// TIA Portal V20 export
FUNCTION_BLOCK "F-FB_Laser"   // FB140, F_LAD
{ S7_Optimized_Access := 'TRUE' }
// stored: AutoNumber false
   VAR
      FDBACK_LaserPowerSupply : FDBACK;
      FDBACK_Shutter : FDBACK;
      sFeedBackShutter : Bool;
      sAckFdbShutter : Bool;
      sLaserSupplyPower : Bool;
      sAckFdbPowLaser : Bool;
      sPositiveFrontButtonShutter : Bool;
      sNegativeFrontMaintenanceDoor : Bool;
      sNegativeFrontDoor : Bool;
      sNegativeRoofLeftDoor : Bool;
      sNegativeRoofRightDoor : Bool;
      sNegativeLaserExternDoor : Bool;
      sNegativeSasOneDoor : Bool;
   END_VAR
   VAR_TEMP   // added for the SCL form of the ladder/FBD networks
      _w1 : Bool;
      _w2 : Bool;
      _w3 : Bool;
      _w4 : Bool;
      _w5 : Bool;
      _w6 : Bool;
      _w7 : Bool;
   END_VAR
BEGIN

REGION Network 1: Laser shutter setting mode, allow opening shutter
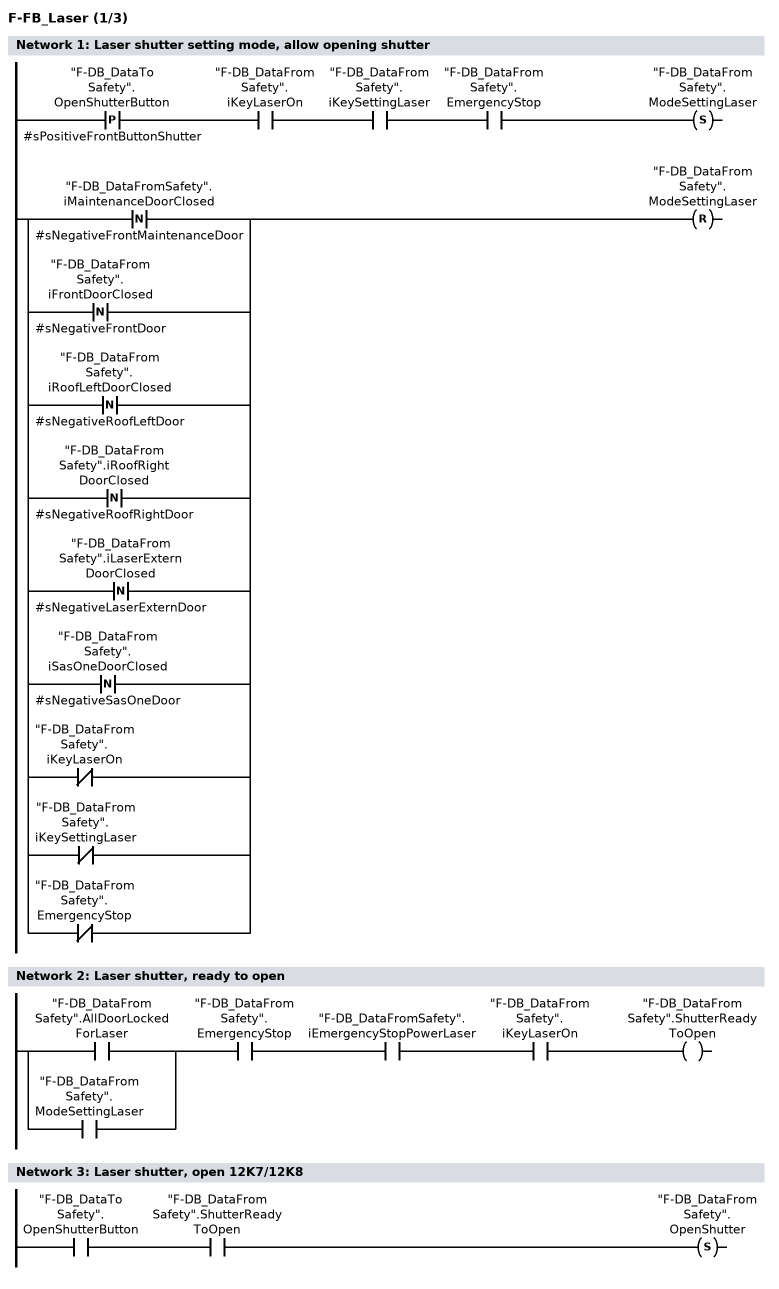
   RUNG wire#powerrail
      P_Contact(operand := "F-DB_DataToSafety".OpenShutterButton, bit := #sPositiveFrontButtonShutter)
      Contact( "F-DB_DataFromSafety".iKeyLaserOn )
      Contact( "F-DB_DataFromSafety".iKeySettingLaser )
      Contact( "F-DB_DataFromSafety".EmergencyStop )
      S_Coil( "F-DB_DataFromSafety".ModeSettingLaser )
   END_RUNG
   RUNG wire#powerrail
      N_Contact(operand := "F-DB_DataFromSafety".iMaintenanceDoorClosed, bit := #sNegativeFrontMaintenanceDoor)
      wire#w1
      R_Coil( "F-DB_DataFromSafety".ModeSettingLaser )
   END_RUNG
   RUNG wire#powerrail
      N_Contact(operand := "F-DB_DataFromSafety".iFrontDoorClosed, bit := #sNegativeFrontDoor)
   END_RUNG wire#w1
   RUNG wire#powerrail
      N_Contact(operand := "F-DB_DataFromSafety".iRoofLeftDoorClosed, bit := #sNegativeRoofLeftDoor)
   END_RUNG wire#w1
   RUNG wire#powerrail
      N_Contact(operand := "F-DB_DataFromSafety".iRoofRightDoorClosed, bit := #sNegativeRoofRightDoor)
   END_RUNG wire#w1
   RUNG wire#powerrail
      N_Contact(operand := "F-DB_DataFromSafety".iLaserExternDoorClosed, bit := #sNegativeLaserExternDoor)
   END_RUNG wire#w1
   RUNG wire#powerrail
      N_Contact(operand := "F-DB_DataFromSafety".iSasOneDoorClosed, bit := #sNegativeSasOneDoor)
   END_RUNG wire#w1
   RUNG wire#powerrail
      I_Contact( "F-DB_DataFromSafety".iKeyLaserOn )
   END_RUNG wire#w1
   RUNG wire#powerrail
      I_Contact( "F-DB_DataFromSafety".iKeySettingLaser )
   END_RUNG wire#w1
   RUNG wire#powerrail
      I_Contact( "F-DB_DataFromSafety".EmergencyStop )
   END_RUNG wire#w1
   // the same network as SCL:
   #_w1 := "F-DB_DataToSafety".OpenShutterButton AND NOT #sPositiveFrontButtonShutter;   // rising edge of "F-DB_DataToSafety".OpenShutterButton
   #sPositiveFrontButtonShutter := "F-DB_DataToSafety".OpenShutterButton;
   IF #_w1 AND "F-DB_DataFromSafety".iKeyLaserOn AND "F-DB_DataFromSafety".iKeySettingLaser AND "F-DB_DataFromSafety".EmergencyStop THEN
       "F-DB_DataFromSafety".ModeSettingLaser := TRUE;
   END_IF;
   #_w2 := NOT "F-DB_DataFromSafety".iMaintenanceDoorClosed AND #sNegativeFrontMaintenanceDoor;   // falling edge of "F-DB_DataFromSafety".iMaintenanceDoorClosed
   #sNegativeFrontMaintenanceDoor := "F-DB_DataFromSafety".iMaintenanceDoorClosed;
   #_w3 := NOT "F-DB_DataFromSafety".iFrontDoorClosed AND #sNegativeFrontDoor;   // falling edge of "F-DB_DataFromSafety".iFrontDoorClosed
   #sNegativeFrontDoor := "F-DB_DataFromSafety".iFrontDoorClosed;
   #_w4 := NOT "F-DB_DataFromSafety".iRoofLeftDoorClosed AND #sNegativeRoofLeftDoor;   // falling edge of "F-DB_DataFromSafety".iRoofLeftDoorClosed
   #sNegativeRoofLeftDoor := "F-DB_DataFromSafety".iRoofLeftDoorClosed;
   #_w5 := NOT "F-DB_DataFromSafety".iRoofRightDoorClosed AND #sNegativeRoofRightDoor;   // falling edge of "F-DB_DataFromSafety".iRoofRightDoorClosed
   #sNegativeRoofRightDoor := "F-DB_DataFromSafety".iRoofRightDoorClosed;
   #_w6 := NOT "F-DB_DataFromSafety".iLaserExternDoorClosed AND #sNegativeLaserExternDoor;   // falling edge of "F-DB_DataFromSafety".iLaserExternDoorClosed
   #sNegativeLaserExternDoor := "F-DB_DataFromSafety".iLaserExternDoorClosed;
   #_w7 := NOT "F-DB_DataFromSafety".iSasOneDoorClosed AND #sNegativeSasOneDoor;   // falling edge of "F-DB_DataFromSafety".iSasOneDoorClosed
   #sNegativeSasOneDoor := "F-DB_DataFromSafety".iSasOneDoorClosed;
   IF #_w2 OR #_w3 OR #_w4 OR #_w5 OR #_w6 OR #_w7 OR NOT "F-DB_DataFromSafety".iKeyLaserOn OR NOT "F-DB_DataFromSafety".iKeySettingLaser OR NOT "F-DB_DataFromSafety".EmergencyStop THEN
       "F-DB_DataFromSafety".ModeSettingLaser := FALSE;
   END_IF;
END_REGION

REGION Network 2: Laser shutter, ready to open
   RUNG wire#powerrail
      Contact( "F-DB_DataFromSafety".AllDoorLockedForLaser )
      wire#w1
      Contact( "F-DB_DataFromSafety".EmergencyStop )
      Contact( "F-DB_DataFromSafety".iEmergencyStopPowerLaser )
      Contact( "F-DB_DataFromSafety".iKeyLaserOn )
      Coil( "F-DB_DataFromSafety".ShutterReadyToOpen )
   END_RUNG
   RUNG wire#powerrail
      Contact( "F-DB_DataFromSafety".ModeSettingLaser )
   END_RUNG wire#w1
   // the same network as SCL:
   "F-DB_DataFromSafety".ShutterReadyToOpen := ("F-DB_DataFromSafety".AllDoorLockedForLaser OR "F-DB_DataFromSafety".ModeSettingLaser) AND "F-DB_DataFromSafety".EmergencyStop AND "F-DB_DataFromSafety".iEmergencyStopPowerLaser AND "F-DB_DataFromSafety".iKeyLaserOn;
END_REGION

REGION Network 3: Laser shutter, open 12K7/12K8
   RUNG wire#powerrail
      Contact( "F-DB_DataToSafety".OpenShutterButton )
      Contact( "F-DB_DataFromSafety".ShutterReadyToOpen )
      S_Coil( "F-DB_DataFromSafety".OpenShutter )
   END_RUNG
   // the same network as SCL:
   IF "F-DB_DataToSafety".OpenShutterButton AND "F-DB_DataFromSafety".ShutterReadyToOpen THEN
       "F-DB_DataFromSafety".OpenShutter := TRUE;
   END_IF;
END_REGION

REGION Network 4: Laser shutter, close
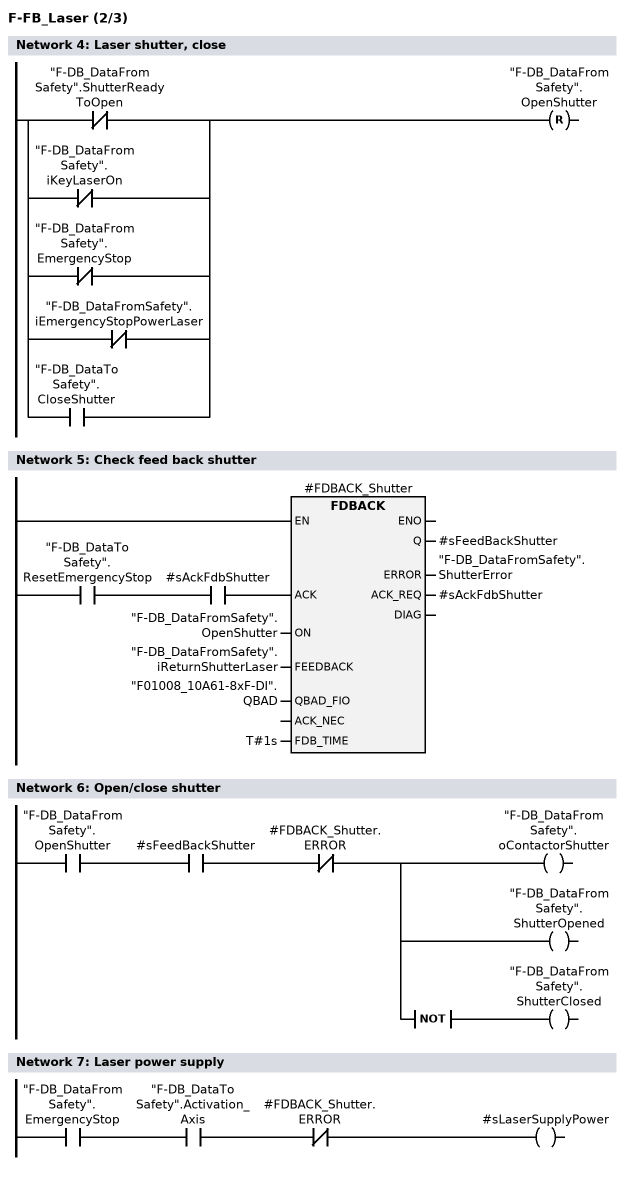
   RUNG wire#powerrail
      I_Contact( "F-DB_DataFromSafety".ShutterReadyToOpen )
      wire#w1
      R_Coil( "F-DB_DataFromSafety".OpenShutter )
   END_RUNG
   RUNG wire#powerrail
      I_Contact( "F-DB_DataFromSafety".iKeyLaserOn )
   END_RUNG wire#w1
   RUNG wire#powerrail
      I_Contact( "F-DB_DataFromSafety".EmergencyStop )
   END_RUNG wire#w1
   RUNG wire#powerrail
      I_Contact( "F-DB_DataFromSafety".iEmergencyStopPowerLaser )
   END_RUNG wire#w1
   RUNG wire#powerrail
      Contact( "F-DB_DataToSafety".CloseShutter )
   END_RUNG wire#w1
   // the same network as SCL:
   IF NOT "F-DB_DataFromSafety".ShutterReadyToOpen OR NOT "F-DB_DataFromSafety".iKeyLaserOn OR NOT "F-DB_DataFromSafety".EmergencyStop OR NOT "F-DB_DataFromSafety".iEmergencyStopPowerLaser OR "F-DB_DataToSafety".CloseShutter THEN
       "F-DB_DataFromSafety".OpenShutter := FALSE;
   END_IF;
END_REGION

REGION Network 5: Check feed back shutter
   RUNG wire#powerrail
      #FDBACK_Shutter.FDBACK(ACK := wire#w1, ON := "F-DB_DataFromSafety".OpenShutter, FEEDBACK := "F-DB_DataFromSafety".iReturnShutterLaser, QBAD_FIO := "F01008_10A61-8xF-DI".QBAD, ACK_NEC :=, FDB_TIME := T#1s, Q => #sFeedBackShutter, ERROR => "F-DB_DataFromSafety".ShutterError, ACK_REQ => #sAckFdbShutter, DIAG =>)
   END_RUNG
   RUNG wire#powerrail
      Contact( "F-DB_DataToSafety".ResetEmergencyStop )
      Contact( #sAckFdbShutter )
   END_RUNG wire#w1
   // the same network as SCL:
   #FDBACK_Shutter(ACK := "F-DB_DataToSafety".ResetEmergencyStop AND #sAckFdbShutter,   // FDBACK
                   ON := "F-DB_DataFromSafety".OpenShutter,
                   FEEDBACK := "F-DB_DataFromSafety".iReturnShutterLaser,
                   QBAD_FIO := "F01008_10A61-8xF-DI".QBAD,
                   FDB_TIME := T#1s,
                   Q => #sFeedBackShutter,
                   ERROR => "F-DB_DataFromSafety".ShutterError,
                   ACK_REQ => #sAckFdbShutter);
END_REGION

REGION Network 6: Open/close shutter
   RUNG wire#powerrail
      Contact( "F-DB_DataFromSafety".OpenShutter )
      Contact( #sFeedBackShutter )
      I_Contact( #FDBACK_Shutter.ERROR )
      wire#w1
      Coil( "F-DB_DataFromSafety".oContactorShutter )
   END_RUNG
   RUNG wire#w1
      Coil( "F-DB_DataFromSafety".ShutterOpened )
   END_RUNG
   RUNG wire#w1
      Not()
      Coil( "F-DB_DataFromSafety".ShutterClosed )
   END_RUNG
   // the same network as SCL:
   "F-DB_DataFromSafety".oContactorShutter := "F-DB_DataFromSafety".OpenShutter AND #sFeedBackShutter AND NOT #FDBACK_Shutter.ERROR;
   "F-DB_DataFromSafety".ShutterOpened := "F-DB_DataFromSafety".oContactorShutter;
   "F-DB_DataFromSafety".ShutterClosed := NOT "F-DB_DataFromSafety".oContactorShutter;
END_REGION

REGION Network 7: Laser power supply
   RUNG wire#powerrail
      Contact( "F-DB_DataFromSafety".EmergencyStop )
      Contact( "F-DB_DataToSafety".Activation_Axis )
      I_Contact( #FDBACK_Shutter.ERROR )
      Coil( #sLaserSupplyPower )
   END_RUNG
   // the same network as SCL:
   #sLaserSupplyPower := "F-DB_DataFromSafety".EmergencyStop AND "F-DB_DataToSafety".Activation_Axis AND NOT #FDBACK_Shutter.ERROR;
END_REGION

REGION Network 8: Check feed back laser power supply
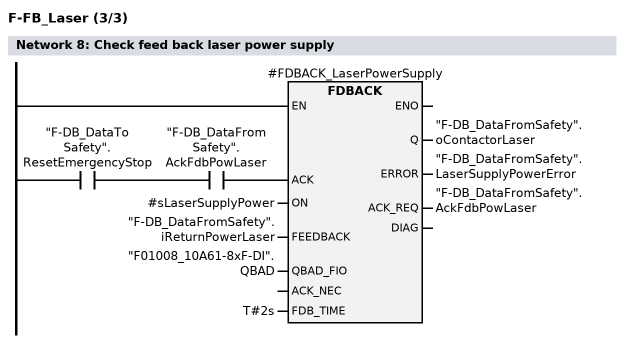
   RUNG wire#powerrail
      #FDBACK_LaserPowerSupply.FDBACK(ACK := wire#w1, ON := #sLaserSupplyPower, FEEDBACK := "F-DB_DataFromSafety".iReturnPowerLaser, QBAD_FIO := "F01008_10A61-8xF-DI".QBAD, ACK_NEC :=, FDB_TIME := T#2s, Q => "F-DB_DataFromSafety".oContactorLaser, ERROR => "F-DB_DataFromSafety".LaserSupplyPowerError, ACK_REQ => "F-DB_DataFromSafety".AckFdbPowLaser, DIAG =>)
   END_RUNG
   RUNG wire#powerrail
      Contact( "F-DB_DataToSafety".ResetEmergencyStop )
      Contact( "F-DB_DataFromSafety".AckFdbPowLaser )
   END_RUNG wire#w1
   // the same network as SCL:
   #FDBACK_LaserPowerSupply(ACK := "F-DB_DataToSafety".ResetEmergencyStop AND "F-DB_DataFromSafety".AckFdbPowLaser,   // FDBACK
                           ON := #sLaserSupplyPower,
                           FEEDBACK := "F-DB_DataFromSafety".iReturnPowerLaser,
                           QBAD_FIO := "F01008_10A61-8xF-DI".QBAD,
                           FDB_TIME := T#2s,
                           Q => "F-DB_DataFromSafety".oContactorLaser,
                           ERROR => "F-DB_DataFromSafety".LaserSupplyPowerError,
                           ACK_REQ => "F-DB_DataFromSafety".AckFdbPowLaser);
END_REGION
END_FUNCTION_BLOCK
